Universal Robots PolyScope program: _adminCG-invBToPHome.urp

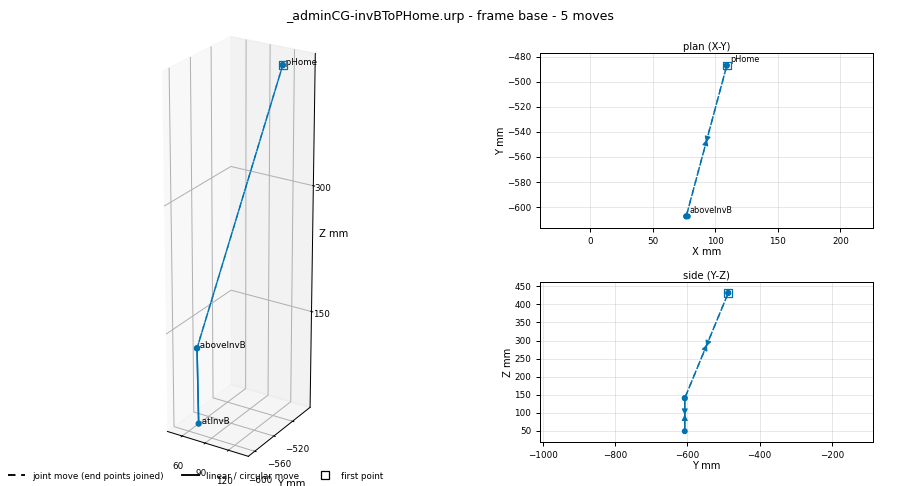
[picture p0: tool path of _adminCG-invBToPHome.urp in frame base, 5 of 5 moves have a stored position in this frame; points joined in program order, loops and branches not executed]
Program _adminCG-invBToPHome (installation=admin directory=/programs/THU_530PM createdIn=3.15.8.106339 lastSavedIn=3.15.8.106339 robotSerialNumber=2015350926)
Calibrated DH parameters: a=[0, -0.425, -0.39225, 0, 0, 0]; d=[0.089159, 0, 0, 0.10915, 0.09465, 0.0823]; alpha=[1.570796, 0, 0, 1.570796, -1.570796, 0]; deltaTheta=[0, 0, 0, 0, 0, 0]
Robot Program (runOnlyOnce=true)
  Call _adminLinearIndex3
  Set DigitalOutput pin=digital_out[0]; digitalValue=0
  MoveJ speed 60 deg/s, acceleration 80 deg/s^2 (useActiveTCP=true)
    Waypoint pHome: TCP in base x=109.141 y=-486.906 z=431.874 mm, rx=0 ry=-3.1416 rz=0.0003 rad; joints [89.999, -90.001, 90.001, -90.01, -90.001, -0.001] deg
    Waypoint aboveInvB: TCP in base x=76.73 y=-607.442 z=140.178 mm, rx=2.2211 ry=2.2214 rz=-0.0003 rad; joints [86.93, -62.051, 100.171, -128.138, -89.997, 86.922] deg
  MoveL speed 250 mm/s, acceleration 1200 mm/s^2 (useActiveTCP=true) feature=Base
    Waypoint atInvB: TCP in base x=78.002 y=-607.451 z=48.551 mm, rx=2.2212 ry=2.2215 rz=-0.0002 rad; joints [87.051, -53.284, 102.949, -139.675, -89.998, 87.044] deg
    Set DigitalOutput pin=digital_out[0]; digitalValue=1
    Wait Sleep waitTime=1
    Waypoint aboveInvB: TCP in base x=76.73 y=-607.442 z=140.178 mm, rx=2.2211 ry=2.2214 rz=-0.0003 rad; joints [86.93, -62.051, 100.171, -128.138, -89.997, 86.922] deg
  MoveJ speed 60 deg/s, acceleration 80 deg/s^2 (useActiveTCP=true)
    Waypoint pHome: TCP in base x=109.141 y=-486.906 z=431.874 mm, rx=0 ry=-3.1416 rz=0.0003 rad; joints [89.999, -90.001, 90.001, -90.01, -90.001, -0.001] deg
SubProgram -> _adminLinearIndex3
SubProgram _adminLinearIndex3 (keepSynchronizedWithDisk=false) programFile=/programs/me345_admin/_adminLinearIndex3.urp
  Folder Move_linear_slide_Index1
    var_1 := False
    Loop While (checkContinuously=false) expression=var_1≟ False
      var_1 := socket_open("10.241.34.44",4001)
    var_3 := 1
    Send := "s r0x24 21"
    Script: socket_send_string(Send)
    Script: socket_send_byte(13)
    Send_Reply := socket_read_string()
    Send := "s r0xca 103936"
    Script: socket_send_string(Send)
    Script: socket_send_byte(13)
    Send_Reply := socket_read_string()
    Send := "t 1"
    Script: socket_send_string(Send)
    Script: socket_send_byte(13)
    Send_Reply := socket_read_string()
    Loop While (checkContinuously=false) expression=var_3≠0
      Send := "g r0xA0"
      Script: socket_send_string(Send)
      Script: socket_send_byte(13)
      var_3 := socket_get_var("v")
      Wait Sleep waitTime=0.1
    Script: socket_close()
    Script: sync()
